//-----------------------------------------------------------------------------------------------------------
// TriggerBox
//
// HAUD
// 17.07.2024
// - init: ALL outputs will be switched of 
// - controlled via ST_TriggerBox
// - position and timestamp based setting of digital output
// - feedback from digital input with timestamp
// - AxisPosition at timestamp as result
//-----------------------------------------------------------------------------------------------------------
FUNCTION_BLOCK FB_TriggerBox EXTENDS FB_Xfc
VAR
  _Ctrl             : REFERENCE TO ARRAY[1..MAX_TRIGGER_BOX] OF ST_CTRL_TRIGGER;
  _State            : REFERENCE TO ARRAY[1..MAX_TRIGGER_BOX] OF ST_STATE_TRIGGER;

  _Input            : POINTER TO ARRAY[1..MAX_TRIGGER_BOX]   OF ST_DC_Input;
  _Output_2252      : POINTER TO ARRAY[1..MAX_TRIGGER_BOX]   OF ST_DC_Output;

  _Index            : UDINT;
  _AxisId           : UDINT;
  _AxisIndex        : UDINT;

  _CtrlLocal        : ST_CTRL_TRIGGER;
  _McDirection      : Tc2_MC2.MC_Direction;

  _eStateProgress   : E_PROGRESS;
  _eResult          : E_PROGRESS;
  _eInit            : E_PROGRESS;

  _rtrigEnable      : Tc2_Standard.R_TRIG;
  _rtrigInit        : Tc2_Standard.R_TRIG;
  _TrigCount        : UDINT := 1; // counter for active index in _stCtrl.TriggerPosition[]

  _CurrentTime      : ULINT;      // current DC time 64 bit
  _CurrentTimeShort : UDINT;      // current DC time 32 bit
  _LatchTime        : UDINT;
  _SwitchTime       : ULINT;      // DC time for output at _stCtrl.TriggerPosition[_TrigCount]
  _SafeCycles       : BYTE := 3;  // cycles needed to get the SwitchTime onto the terminal/output

  _bError           : BOOL;
  _stMsg            : ST_Message;
  _MessageLevel     : E_MessageType;
END_VAR

PROPERTY Ctrl : REFERENCE TO ARRAY [1..MAX_TRIGGER_BOX] OF ST_CTRL_TRIGGER
SET
_Ctrl REF= Ctrl;
END_SET
END_PROPERTY

METHOD Cycle : BOOL
VAR_INPUT
END_VAR
//-----------------------------------------------------------------------------
// trigger detection
//-----------------------------------------------------------------------------
_rtrigEnable(CLK                := _Ctrl[_Index].Control.Enable);
_rtrigInit(  CLK                := _Ctrl[_Index].Control.Init);
//-----------------------------------------------------------------------------
// forced init
//-----------------------------------------------------------------------------
IF _rtrigInit.Q THEN _eInit     := E_PROGRESS.PROGRESS_INVALID; END_IF
//-----------------------------------------------------------------------------
// clear state
//-----------------------------------------------------------------------------
IF NOT _Ctrl[_Index].Control.Enable 
THEN 
  _eStateProgress               := E_PROGRESS.PROGRESS_INVALID;

  _State[_Index].State          := TO_UINT(_eStateProgress);
END_IF

_eDeviceFunction                := e_Device.XfcTriggerBox + _Index;

_CurrentTime                    := Tc2_EtherCAT.F_GetCurDcTaskTime64();
_CurrentTimeShort               := TO_UDINT(_CurrentTime AND 16#FFFFFFFF);

_State[_Index].Init             := TO_UINT(_eInit);

IF NOT (_eInit = E_PROGRESS.PROGRESS_DONE)
THEN
  _eInit                        := Init();
  RETURN;
END_IF
//-----------------------------------------------------------------------------
// TriggerBox execution
//-----------------------------------------------------------------------------
CASE _eStateProgress
OF
  E_PROGRESS.PROGRESS_INVALID:  // check input data
    IF _rtrigEnable.Q
    THEN
      _State[_Index].State      := TO_UINT(E_PROGRESS.PROGRESS_BUSY);

      _bError                   := FALSE;
      _TrigCount                := 1;     // initialize trigger counter for output on TriggerPositions
      _eStateProgress           := E_PROGRESS.PROGRESS_INIT;

      _CtrlLocal                := _Ctrl[_Index];
      _AxisId                   := _CtrlLocal.AxisId;
      _AxisIndex                := GetIndex(_AxisId);

      _eResult                  := TimeToPosition(FALSE, _AxisId, 0.0, _MessageLevel);
      _eResult                  := WaitForPosition(FALSE, _AxisId, _CtrlLocal.TriggerPosition[_TrigCount], _MessageLevel);

      IF NOT (_AxisIndex > 0) OR NOT (_AxisId > 0)
      THEN
        _bError                 := TRUE;
        _stMsg.iErrorNumber     := 10;
        _stMsg.eSubdevice       := XfcTriggerStart;
        _stMsg.sText            := 'AxisId Invalid ';
        _eStateProgress         := E_PROGRESS.PROGRESS_STILL_WORKING;
      END_IF

      IF NOT (_CtrlLocal.TriggerCount > 0) OR
         NOT (_CtrlLocal.TriggerCount < TO_UDINT(MAX_TRIGGER_COUNT+1))
      THEN
        _bError                 := TRUE;
        _stMsg.iErrorNumber     := 11;
        _stMsg.eSubdevice       := XfcTriggerStart;
        _stMsg.sText            := 'TriggerCount Invalid ';
        _eStateProgress         := E_PROGRESS.PROGRESS_STILL_WORKING;
      END_IF

      IF (_MessageLevel = E_MessageType.eMessageVerbose)
      THEN
        _stMsg.eType            := E_MessageType.eMessageVerbose;
        _stMsg.eDevice          := _eDeviceFunction;
        _stMsg.eSubdevice       := e_Subdevice.XfcTriggerStart;
        _stMsg.iErrorNumber     := _CurrentTime;
        _stMsg.sText            := concat(TO_STRING(_eStateProgress), ': ');
        _stMsg.sText            := concat(_stMsg.sText, TO_STRING(e_Device.XfcAxis));
        _stMsg.sText            := concat(_stMsg.sText, '_ID_');
        _stMsg.sText            := concat(_stMsg.sText, TO_STRING(_AxisId));

        f_MessageSet(_stMsg);
      END_IF
    END_IF


  E_PROGRESS.PROGRESS_INIT:
    _eDeviceAxis                := e_Device.XfcAxis + (_CtrlLocal.AxisId);
    _eResult                    := WaitForPosition(TRUE, _AxisId, _CtrlLocal.TriggerPosition[_TrigCount], _MessageLevel);

    IF (_eResult = E_PROGRESS.PROGRESS_ERROR)
    THEN
      _bError                   := TRUE;
      _stMsg.iErrorNumber       := 16;
      _stMsg.eSubdevice         := XfcWaitForPosition;
      _stMsg.sText              := 'Position not reachable ';
      _eStateProgress           := E_PROGRESS.PROGRESS_STILL_WORKING;

    ELSIF (_eResult = E_PROGRESS.PROGRESS_DONE)
    THEN
      _eStateProgress           := E_PROGRESS.PROGRESS_BUSY;

      IF (_MessageLevel = E_MessageType.eMessageVerbose)
      THEN
        _stMsg.eType            := E_MessageType.eMessageVerbose;
        _stMsg.eDevice          := _eDeviceFunction;
        _stMsg.eSubdevice       := e_Subdevice.XfcWaitForPosition;
        _stMsg.iErrorNumber     := _CurrentTime;
        _stMsg.sText            := concat(TO_STRING(_eStateProgress), ': ');
        _stMsg.sText            := concat(_stMsg.sText, TO_STRING(_XfcDurationToPosition[_AxisIndex]));

        f_MessageSet(_stMsg);
      END_IF
    END_IF
END_CASE
//-----------------------------------------------------------------------------
//-----------------------------------------------------------------------------
CASE _eStateProgress
OF
  E_PROGRESS.PROGRESS_BUSY:
    _eResult                    := TimeToPosition(TRUE, _AxisId, _CtrlLocal.TriggerPosition[_TrigCount], _MessageLevel);

    IF (_eResult = E_PROGRESS.PROGRESS_ERROR)
    THEN
      TimeToPosition(FALSE, _AxisId, _CtrlLocal.TriggerPosition[_TrigCount], _MessageLevel);

      _bError                   := TRUE;
      _stMsg.iErrorNumber       := 15;
      _stMsg.sText              := concat('Get TimeToPosition ', TO_STRING(_CtrlLocal.TriggerPosition[_TrigCount]));
      _stMsg.sText              := concat(_stMsg.sText, ' ');
      _eStateProgress           := E_PROGRESS.PROGRESS_STILL_WORKING;

    ELSIF (_eResult = E_PROGRESS.PROGRESS_DONE)
    THEN
      TimeToPosition(FALSE, _AxisId, _CtrlLocal.TriggerPosition[_TrigCount], _MessageLevel);

      _SwitchTime               := _CurrentTime + TO_ULINT(_XfcDurationToPosition[_AxisIndex]);
      _eResult                  := SwitchOn_2252(FALSE, _SwitchTime, 3);
 
      IF (_MessageLevel = E_MessageType.eMessageVerbose)
      THEN
        _stMsg.eType            := E_MessageType.eMessageVerbose;
        _stMsg.eDevice          := _eDeviceFunction;
        _stMsg.eSubdevice       := e_Subdevice.XfcTimeToPosition;
        _stMsg.iErrorNumber     := _SwitchTime;
        _stMsg.sText            := concat(TO_STRING(_eStateProgress), ': ');
        _stMsg.sText            := concat(_stMsg.sText, TO_STRING(_XfcDurationToPosition[_AxisIndex]));

        f_MessageSet(_stMsg);
      END_IF
      _eStateProgress           := E_PROGRESS.PROGRESS_PREPARE;
    END_IF
END_CASE
//-----------------------------------------------------------------------------
//-----------------------------------------------------------------------------
CASE _eStateProgress
OF
  E_PROGRESS.PROGRESS_PREPARE:
    //_State[_Index].State        := TO_UINT(_eState);
    _eResult                    := SwitchOn_2252(TRUE, _SwitchTime, 3);


    IF (_CtrlLocal.Control.NoFeedback)
    THEN
      IF (_eResult = E_PROGRESS.PROGRESS_ERROR)
      THEN
        _bError                 := TRUE;
        _stMsg.iErrorNumber     := 12;
        _stMsg.eSubdevice       := XfcSwitchOn_2252;
        _stMsg.sText            := 'NO_FEEDBACK: Switch Time in the past ';
        _eStateProgress         := E_PROGRESS.PROGRESS_STILL_WORKING;

      ELSIF (_eResult = E_PROGRESS.PROGRESS_DONE)
      THEN
        _eStateProgress         := E_PROGRESS.PROGRESS_CHECK;
      END_IF

    ELSIF (_eResult = E_PROGRESS.PROGRESS_ERROR)
    THEN
        _bError                 := TRUE;
        _stMsg.iErrorNumber     := 13;
        _stMsg.eSubdevice       := XfcSwitchOn_2252;
        _stMsg.sText            := 'Switch Time in the past ';
        _eStateProgress         := E_PROGRESS.PROGRESS_STILL_WORKING;
    END_IF

    IF (_Input^[_Index].Input) OR
       (_Input^[_Index].LatchPositive >= _SwitchTime)
    THEN
      _LatchTime                := TO_UDINT(_Input^[_Index].LatchPositive AND 16#FFFFFFFF);

      IF (_MessageLevel = E_MessageType.eMessageVerbose)
      THEN
        _stMsg.eType            := E_MessageType.eMessageVerbose;
        _stMsg.eDevice          := _eDeviceFunction;
        _stMsg.eSubdevice       := e_Subdevice.XfcLatchPosition;
        _stMsg.iErrorNumber     := _LatchTime;
        _stMsg.sText            := concat(TO_STRING(_eStateProgress), ': ');
        _stMsg.sText            := concat(_stMsg.sText, TO_STRING(_eDeviceAxis));

        f_MessageSet(_stMsg);
      END_IF
      _eStateProgress           := E_PROGRESS.PROGRESS_STARTUP;
      _eResult                  := PositionAtTime(FALSE, _CtrlLocal.AxisId, 0, _MessageLevel);
      _eResult                  := SwitchOn_2252(FALSE, _SwitchTime, 3);
    END_IF
END_CASE
//-----------------------------------------------------------------------------
//-----------------------------------------------------------------------------
CASE _eStateProgress
OF
  E_PROGRESS.PROGRESS_STARTUP:
    //_State[_Index].State        := TO_UINT(_eState);
    _eResult                    := PositionAtTime(TRUE, _CtrlLocal.AxisId, _LatchTime, _MessageLevel);

    IF (_eResult = E_PROGRESS.PROGRESS_ERROR)
    THEN
      _bError                   := TRUE;
      _stMsg.iErrorNumber       := 14;
      _stMsg.sText              := 'PositionAtTime LatchPositive ';
      _eStateProgress           := E_PROGRESS.PROGRESS_STILL_WORKING;
      _eResult                  := PositionAtTime(FALSE, _CtrlLocal.AxisId, 0, _MessageLevel);

    ELSIF (_eResult = E_PROGRESS.PROGRESS_DONE)
    THEN
      _State[_Index].FlashPosition[_TrigCount]  := _XfcRecordedPosition[_AxisIndex];

      IF (_MessageLevel = E_MessageType.eMessageVerbose)
      THEN
        _stMsg.eType            := E_MessageType.eMessageVerbose;
        _stMsg.eDevice          := _eDeviceFunction;
        _stMsg.eSubdevice       := e_Subdevice.XfcRecordedPosition;
        _stMsg.iErrorNumber     := _LatchTime;
        _stMsg.sText            := concat(TO_STRING(_eStateProgress), ': ');
        _stMsg.sText            := concat(_stMsg.sText, TO_STRING(_XfcRecordedPosition[_AxisIndex]));

        f_MessageSet(_stMsg);
      END_IF
      _eStateProgress           := E_PROGRESS.PROGRESS_CHECK;
      _eResult                  := PositionAtTime(FALSE, _CtrlLocal.AxisId, 0, _MessageLevel);
      _eResult                  := SwitchOff_2252(FALSE, 3);
    END_IF
END_CASE
//-----------------------------------------------------------------------------
//-----------------------------------------------------------------------------
CASE _eStateProgress
OF
  E_PROGRESS.PROGRESS_CHECK:
    _State[_Index].State        := TO_UINT(_eStateProgress) + TO_UINT(_TrigCount);
    _eResult                    := SwitchOff_2252(TRUE, 4);
    IF (_eResult = E_PROGRESS.PROGRESS_DONE)
    THEN
      _eResult                  := SwitchOff_2252(FALSE, 4);
      _TrigCount                := _TrigCount + 1;

      IF (_TrigCount > _CtrlLocal.TriggerCount)
      THEN
        _eStateProgress         := E_PROGRESS.PROGRESS_OCCUPIED;
      ELSE
        _eStateProgress         := E_PROGRESS.PROGRESS_INIT;
        _eResult                := WaitForPosition(FALSE, _AxisId, _CtrlLocal.TriggerPosition[_TrigCount], _MessageLevel);
      END_IF
    END_IF
END_CASE
//-----------------------------------------------------------------------------
//-----------------------------------------------------------------------------
CASE _eStateProgress
OF
  E_PROGRESS.PROGRESS_OCCUPIED:
    _eStateProgress             := E_PROGRESS.PROGRESS_WORKING;
END_CASE
//-----------------------------------------------------------------------------
//-----------------------------------------------------------------------------
CASE _eStateProgress
OF
  E_PROGRESS.PROGRESS_WORKING:
    _eStateProgress             := E_PROGRESS.PROGRESS_STILL_WORKING;
END_CASE
//-----------------------------------------------------------------------------
//-----------------------------------------------------------------------------
CASE _eStateProgress
OF
  E_PROGRESS.PROGRESS_STILL_WORKING:
    IF NOT _bError
    THEN
      _eStateProgress           := E_PROGRESS.PROGRESS_DONE;

      IF (_MessageLevel > E_MessageType.eMessageWarning)
      THEN
        _stMsg.eType            := E_MessageType.eMessageInfo;
        _stMsg.eDevice          := _eDeviceFunction;
        _stMsg.eSubdevice       := e_Subdevice.XfcTriggerOut;
        _stMsg.iErrorNumber     := _CurrentTime;
        _stMsg.sText            := concat(TO_STRING(_eStateProgress), ': ');
        _stMsg.sText            := concat(_stMsg.sText, TO_STRING(e_Device.XfcAxis));
        _stMsg.sText            := concat(_stMsg.sText, '_ID_');
        _stMsg.sText            := concat(_stMsg.sText, TO_STRING(_AxisId));
        f_MessageSet(_stMsg);
      END_IF
      _State[_Index].State      := TO_UINT(_eStateProgress);
    ELSE
      _eStateProgress           := E_PROGRESS.PROGRESS_ERROR;

      _stMsg.eType              := E_MessageType.eMessageError;
      _stMsg.eDevice            := _eDeviceFunction;
      _stMsg.eSubdevice         := e_Subdevice.XfcTriggerOut;
      _stMsg.sText              := concat(_stMsg.sText, TO_STRING(_eStateProgress));

      f_MessageSet(_stMsg);

      _State[_Index].State      := TO_UINT(_eStateProgress) + TO_UINT(_stMsg.iErrorNumber);
    END_IF
END_CASE
END_METHOD

PROPERTY Index : udint
GET
Index := _Index;
END_GET
SET
_Index := Index;
END_SET
END_PROPERTY

METHOD Init : E_PROGRESS
VAR_INST
  _eState         : E_PROGRESS;
  _eResult        : E_PROGRESS;

  _stMsg          : ST_Message;
  _bError         : BOOL;
  _udiErrorId     : UDINT;

  _nIdx           : udint;
END_VAR

_stMsg.eDevice                  := _eDeviceFunction;
_stMsg.eSubdevice               := XfcInit;


CASE _eInit
OF
  E_PROGRESS.PROGRESS_INVALID:
    _eState                     := E_PROGRESS.PROGRESS_INIT;
    _bError                     := FALSE;
    _udiErrorId                 := 0;
END_CASE
//-----------------------------------------------------------------------------
//-----------------------------------------------------------------------------
CASE _eState
OF
  E_PROGRESS.PROGRESS_INIT:
    _eResult                    := SwitchOff_2252(FALSE, 2);
    _eState                     := E_PROGRESS.PROGRESS_BUSY;

      IF (_MessageLevel = E_MessageType.eMessageVerbose)
      THEN
        _stMsg.eType            := E_MessageType.eMessageVerbose;
        _stMsg.iErrorNumber     := 0;
        _stMsg.sText            := TO_STRING(_eState);

        f_MessageSet(_stMsg);
      END_IF

  //-----------------------------------------------------------------------------
  // clear output terminals 2252
  //-----------------------------------------------------------------------------
  E_PROGRESS.PROGRESS_BUSY:
    _eResult                    := SwitchOff_2252(TRUE, 10);

    IF (_eResult = E_PROGRESS.PROGRESS_DONE)
    THEN
      IF (_Index > 0) AND
         (_Index < MAX_TRIGGER_BOX+1)
      THEN
        FOR _nIdx := 1 TO MAX_TRIGGER_COUNT
        DO
          _State[_Index].FlashPosition[_nIdx] := 0.0;
        END_FOR
      END_IF

      _eState                   := E_PROGRESS.PROGRESS_PREPARE;
      _eResult                  := SwitchOff_2252(FALSE, 10);
    END_IF
END_CASE
//-----------------------------------------------------------------------------
// reserve states for future timestamp outputs with dedicated switch off
//-----------------------------------------------------------------------------
CASE _eState
OF
  E_PROGRESS.PROGRESS_PREPARE:
    _eState                     := E_PROGRESS.PROGRESS_STARTUP;
END_CASE
//-----------------------------------------------------------------------------
//-----------------------------------------------------------------------------
CASE _eState
OF
  E_PROGRESS.PROGRESS_STARTUP:
    _eState                     := E_PROGRESS.PROGRESS_CHECK;
END_CASE
//-----------------------------------------------------------------------------
//-----------------------------------------------------------------------------
CASE _eState
OF
  E_PROGRESS.PROGRESS_CHECK:
    _eState                     := E_PROGRESS.PROGRESS_OCCUPIED;
END_CASE
//-----------------------------------------------------------------------------
//-----------------------------------------------------------------------------
CASE _eState
OF
  E_PROGRESS.PROGRESS_OCCUPIED:
    _eState                     := E_PROGRESS.PROGRESS_WORKING;
END_CASE
//-----------------------------------------------------------------------------
//-----------------------------------------------------------------------------
CASE _eState
OF
  E_PROGRESS.PROGRESS_WORKING:
    _eState                     := E_PROGRESS.PROGRESS_STILL_WORKING;
END_CASE
//-----------------------------------------------------------------------------
//-----------------------------------------------------------------------------
CASE _eState
OF
  E_PROGRESS.PROGRESS_STILL_WORKING:
    IF NOT _bError
    THEN
      _eState                   := E_PROGRESS.PROGRESS_DONE;

      IF (_MessageLevel > E_MessageType.eMessageWarning)
      THEN
        _stMsg.eType            := E_MessageType.eMessageInfo;
        _stMsg.iErrorNumber     := 0;
        _stMsg.sText            := TO_STRING(_eState);
      END_IF
    ELSE
      _eState                   := E_PROGRESS.PROGRESS_ERROR;

      _stMsg.eType              := E_MessageType.eMessageError;
      _stMsg.iErrorNumber       := _udiErrorId;
      _stMsg.sText              := TO_STRING(_eState);
    END_IF
END_CASE

Init                            := _eState;
END_METHOD

PROPERTY Input : pointer TO ARRAY [1..MAX_TRIGGER_BOX] OF ST_DC_Input
SET
_Input := Input;
END_SET
END_PROPERTY

PROPERTY MessageLevel : e_messagetype
GET
MessageLevel := _MessageLevel;
END_GET
SET
_MessageLevel := MessageLevel;
END_SET
END_PROPERTY

PROPERTY Output_2252 : pointer TO ARRAY [1..MAX_TRIGGER_BOX] OF ST_DC_Output
SET
_Output_2252 := Output_2252;
END_SET
END_PROPERTY

PROPERTY State : REFERENCE TO ARRAY[1..MAX_TRIGGER_BOX] OF ST_STATE_TRIGGER
SET
_State REF= State;
END_SET
END_PROPERTY

METHOD SwitchOff_2252 : E_PROGRESS
VAR_INPUT
  Execute         : BOOL;
  DurationCycles  : UINT := 3;   // PLC cycles are counted after the output time was reached before the method returns done
END_VAR
VAR_INST
  _bError             : BOOL;
  _eState             : E_PROGRESS;

  _stMsg              : ST_Message;
  _CurrentStartTime   : ULINT;
  _nCount             : UINT;
END_VAR
IF NOT Execute THEN _eState     := E_PROGRESS.PROGRESS_INIT;  END_IF


CASE _eState
OF
  E_PROGRESS.PROGRESS_INIT:
    IF Execute
    THEN
      _nCount                   := 0;
      _bError                   := FALSE;
      _eState                   := E_PROGRESS.PROGRESS_BUSY;
      _CurrentStartTime         := Tc2_EtherCAT.F_GetCurDcTaskTime64();

      _Output_2252^[_Index].nActivate     := 0;

      IF (_MessageLevel = E_MessageType.eMessageVerbose)
      THEN
        _stMsg.eType            := E_MessageType.eMessageVerbose;
        _stMsg.eDevice          := _eDeviceFunction;
        _stMsg.eSubdevice       := XfcSwitchOff_2252;
        _stMsg.iErrorNumber     := _CurrentStartTime;
        _stMsg.sText            := TO_STRING(_eState);
        f_MessageSet(_stMsg);
      END_IF
    END_IF

  E_PROGRESS.PROGRESS_BUSY:
    _Output_2252^[_Index].Ch1_Output    := FALSE;
    _Output_2252^[_Index].Ch2_Output    := FALSE;

    _Output_2252^[_Index].Ch1_Tristate  := FALSE;
    _Output_2252^[_Index].Ch2_Tristate  := FALSE;

    _Output_2252^[_Index].dcStartTime   := (_CurrentStartTime + DurationCycles*2_000_000);
    _Output_2252^[_Index].nActivate     := 0;
    _eState                                 := E_PROGRESS.PROGRESS_PREPARE;


  E_PROGRESS.PROGRESS_PREPARE:
    _Output_2252^[_Index].nActivate     := 3;
    _eState                                 := E_PROGRESS.PROGRESS_STARTUP;

  E_PROGRESS.PROGRESS_STARTUP:
    IF (_CurrentTime > _Output_2252^[_Index].dcStartTime)
    THEN
      //_Output_2252^[_Index].nActivate   := 0;
      _eState                               := E_PROGRESS.PROGRESS_CHECK;
    END_IF

  E_PROGRESS.PROGRESS_CHECK:
    _nCount                                 := _nCount + 1;
    IF (_nCount > DurationCycles-1)
    THEN
      _Output_2252^[_Index].nActivate   := 0;
      _eState                               := E_PROGRESS.PROGRESS_STILL_WORKING;
    END_IF
END_CASE
//-----------------------------------------------------------------------------
//-----------------------------------------------------------------------------
CASE _eState
OF
  E_PROGRESS.PROGRESS_STILL_WORKING:
    IF NOT _bError
    THEN
      _eState                   := E_PROGRESS.PROGRESS_DONE;
      IF (_MessageLevel > E_MessageType.eMessageWarning)
      THEN
        _stMsg.eType            := E_MessageType.eMessageInfo;
        _stMsg.eDevice          := _eDeviceFunction;
        _stMsg.eSubdevice       := XfcSwitchOff_2252;
        _stMsg.iErrorNumber     := _CurrentTime;
        _stMsg.sText            := TO_STRING(_eState);
        f_MessageSet(_stMsg);
      END_IF
    ELSE
      _eState                   := E_PROGRESS.PROGRESS_ERROR;

      _stMsg.eType              := E_MessageType.eMessageError;
      _stMsg.eDevice            := _eDeviceFunction;
      _stMsg.eSubdevice         := XfcSwitchOff_2252;
      _stMsg.sText              := concat(_stMsg.sText, TO_STRING(_eState));

      f_MessageSet(_stMsg);
 
    END_IF
END_CASE


SwitchOff_2252                  := _eState;
END_METHOD

METHOD SwitchOn_2252 : E_PROGRESS // uses _Output[] datafield directly
VAR_INPUT
  Execute         : BOOL;
  StartTime       : ULINT;
  DurationCycles  : UINT := 3;   // PLC cycles are counted after the output time was reached before the method returns done
END_VAR
VAR_INST
  _bError             : BOOL;
  _eState             : E_PROGRESS;

  _stMsg              : ST_Message;
  _CurrentStartTime   : ULINT;
  _nCount             : UINT;
END_VAR
IF NOT Execute THEN _eState     := E_PROGRESS.PROGRESS_INIT;  END_IF


CASE _eState
OF
  E_PROGRESS.PROGRESS_INIT:
    IF Execute
    THEN
      _nCount                   := 0;
      _bError                   := FALSE;
      _eState                   := E_PROGRESS.PROGRESS_BUSY;
      _CurrentStartTime         := Tc2_EtherCAT.F_GetCurDcTaskTime64();

      IF (_MessageLevel = E_MessageType.eMessageVerbose)
      THEN
        _stMsg.eType            := E_MessageType.eMessageVerbose;
        _stMsg.eDevice          := _eDeviceFunction;
        _stMsg.eSubdevice       := XfcSwitchOn_2252;
        _stMsg.iErrorNumber     := _CurrentStartTime;
        _stMsg.sText            := TO_STRING(_eState);
        f_MessageSet(_stMsg);
      END_IF

      IF NOT ((_CurrentStartTime + _SafeCycles*1_000_000) < StartTime)
      THEN
        _bError                 := TRUE;
        _stMsg.sText            := 'StartTime too close to CurrentTime ';
        _eState                 := E_PROGRESS.PROGRESS_STILL_WORKING;
      END_IF

    END_IF
END_CASE
//-----------------------------------------------------------------------------
//-----------------------------------------------------------------------------
CASE _eState
OF
  E_PROGRESS.PROGRESS_BUSY:
    _Output_2252^[_Index].Ch1_Output    := TRUE;
    _Output_2252^[_Index].Ch2_Output    := TRUE;

    _Output_2252^[_Index].Ch1_Tristate  := FALSE;
    _Output_2252^[_Index].Ch2_Tristate  := FALSE;

    _Output_2252^[_Index].dcStartTime   := StartTime;
    _Output_2252^[_Index].nActivate     := 0;
    _eState                                 := E_PROGRESS.PROGRESS_PREPARE;


  E_PROGRESS.PROGRESS_PREPARE:
    _Output_2252^[_Index].nActivate     := 3;
    _eState                                 := E_PROGRESS.PROGRESS_CHECK;
END_CASE
//-----------------------------------------------------------------------------
//-----------------------------------------------------------------------------
CASE _eState
OF
  E_PROGRESS.PROGRESS_STARTUP:
    IF (_CurrentTime > StartTime)
    THEN
      _Output_2252^[_Index].nActivate   := 0;
      _eState                               := E_PROGRESS.PROGRESS_CHECK;
    END_IF
END_CASE
//-----------------------------------------------------------------------------
//-----------------------------------------------------------------------------
CASE _eState
OF
  E_PROGRESS.PROGRESS_CHECK:
    _nCount                                 := _nCount + 1;
    IF (_nCount > DurationCycles-1)
    THEN
      _eState                               := E_PROGRESS.PROGRESS_STILL_WORKING;
    END_IF
END_CASE
//-----------------------------------------------------------------------------
//-----------------------------------------------------------------------------
CASE _eState
OF
  E_PROGRESS.PROGRESS_STILL_WORKING:
    IF NOT _bError
    THEN
      _eState                   := E_PROGRESS.PROGRESS_DONE;
      IF (_MessageLevel > E_MessageType.eMessageWarning)
      THEN
        _stMsg.eType            := E_MessageType.eMessageInfo;
        _stMsg.eDevice          := _eDeviceFunction;
        _stMsg.eSubdevice       := XfcSwitchOn_2252;
        _stMsg.iErrorNumber     := _CurrentTime;
        _stMsg.sText            := TO_STRING(_eState);
        f_MessageSet(_stMsg);
      END_IF
    ELSE
      _eState                   := E_PROGRESS.PROGRESS_ERROR;

      _stMsg.eType              := E_MessageType.eMessageError;
      _stMsg.eDevice            := _eDeviceFunction;
      _stMsg.eSubdevice         := XfcSwitchOn_2252;
      _stMsg.sText              := concat(_stMsg.sText, TO_STRING(_eState));

      f_MessageSet(_stMsg);
 
    END_IF
END_CASE


SwitchOn_2252                   := _eState;
END_METHOD

END_FUNCTION_BLOCK

(* stored: Version 1.1.0.1, ProductVersion 3.1.4024.13
   POU FB_TriggerBox: Id {db4923bf-bc34-4aee-8591-dc86a23ff7f9}, SpecialFunc None
   Folder methods: Id {66960e94-618b-4a51-8fe4-7cb0e0c8b66b}
   Folder properties: Id {e525154d-dd27-4c88-81c0-6d06259e3a2a}
   Property Ctrl: Id {5df0cab9-0783-4ce9-b03c-a84423388261}
   Set Set: Id {ad9fa7f7-8ca0-4982-bf1c-b06712bc7c22}
   Method Cycle: Id {0c59e9a7-6d7f-43a4-bd21-5d8b0de0630e}
   Property Index: Id {3c03046a-745d-4156-ad36-4ca380452463}
   Get Get: Id {5bf1b6a3-d598-4816-b77f-32ca015b57dd}
   Set Set: Id {3abce8f0-db48-4c0f-97e9-5137929148c3}
   Method Init: Id {9ed0687f-e23c-4170-9864-3d5c86179885}
   Property Input: Id {6d5ea1b3-e047-43d0-bad1-f57a4f879cb3}
   Set Set: Id {75be905b-dcd0-4597-a76a-347fe44f7078}
   Property MessageLevel: Id {4d136669-d80f-447f-b466-594c0abfb41f}
   Get Get: Id {6cb87e47-382b-4e62-99c5-ef325467f8bb}
   Set Set: Id {2f2e6644-0a3c-4a37-96e1-3cc9898015e3}
   Property Output_2252: Id {e15669ef-9058-4d88-84b4-da3acbfd606a}
   Set Set: Id {3a2d407e-dd79-4982-97d2-461ba1df92d7}
   Property State: Id {b6b3ed77-60e1-45c9-94e8-931cbb2fbd11}
   Set Set: Id {bdd2e01c-0ec2-4c9a-8e6c-460cc0d8b62b}
   Method SwitchOff_2252: Id {41db8b4f-3857-4c1c-92e8-de062d51d11b}
   Method SwitchOn_2252: Id {ea3bc18f-a84f-4d7c-91e2-e60c1c26ddb5} *)
